Universal Robots URScript: 00B_01_JieXian_ToYuBei.script

def P00B_01_JieXian_ToYuBei():
  set_tcp(p[-0.06448999999999999,0.0207,0.28314999999999996,0.0,0.0,1.5902])
  set_payload(0.0)
  set_gravity([0.0, 0.0, 9.82])
  set_standard_analog_input_domain(0, 1)
  set_standard_analog_input_domain(1, 1)
  set_tool_analog_input_domain(0, 1)
  set_tool_analog_input_domain(1, 1)
  set_analog_outputdomain(0, 0)
  set_analog_outputdomain(1, 0)
  set_tool_voltage(0)
  set_input_actions_to_default()
  set_safety_mode_transition_hardness(1)
  $ 1 "机器人程序"
  $ 2 "MoveJ"
  $ 3 "路点_1"
  set_tcp(p[-0.06448999999999999,0.0207,0.28314999999999996,0.0,0.0,1.5902])
  movej(get_inverse_kin(p[.126972404436, .084113536439, .682395636639, .053159442184, -.000755061600, .974100921515], qnear=[1.627946138381958, 0.05497241020202637, -2.831463638936178, -1.8879388014422815, -1.5482295195208948, 2.4669880867004395]), a=0.6981317007977318, v=0.5235987755982988)
  $ 4 "路点_2"
  set_tcp(p[-0.06448999999999999,0.0207,0.28314999999999996,0.0,0.0,1.5902])
  movej(get_inverse_kin(p[.434265315782, .698418251309, .586887469546, -.148324881568, -.158054058472, -1.506931618802], qnear=[1.258681058883667, -1.862976376210348, -2.07282001176943, -0.959076229725973, -1.6494725386248987, 1.3392424583435059]), a=0.6981317007977318, v=0.5235987755982988)
end
